// TwinCAT 3 PLC project Nepionic_Log_Test
// ProgramVersion: 3.1.4026.22
// libraries:
//   [Nepionic_Log], * (Nepionic)
//   [Nepionic_Log_OTel], * (Nepionic)
//   [Nepionic_Log_Syslog], * (Nepionic)
//   Tc2_Standard, * (Beckhoff Automation GmbH)
//   Tc2_System, * (Beckhoff Automation GmbH)
//   Tc2_Utilities, * (Beckhoff Automation GmbH)
//   TcUnit, * (www.tcunit.org)
//   Tc3_Module, * (Beckhoff Automation GmbH)
// project tree:
//   Lib/ LogTester.TcPOU (not stored)
//   Tests/ FB_Test_OTelLogAppender.TcPOU
//   Programs/ TestRunner.TcPOU
//   Tasks/ TestTask.TcTTO (not stored)
// real-time tasks:
//   TASK TestTask: cycle T#10ms, priority 20, ADS port 350

// ---- Tests/FB_Test_OTelLogAppender.TcPOU
/// TcUnit tests for OTelLogAppender.
/// Exercises ring slot writes, head advancement, sequence tagging,
/// severity mapping, attribute storage, ring wrap, and overflow counter.
FUNCTION_BLOCK FB_Test_OTelLogAppender EXTENDS TcUnit.FB_TestSuite
VAR
END_VAR

Test_HeadIncrements();
Test_SequenceCommitted();
Test_SlotContents();
Test_SeverityMapping();
Test_SlotAttrs();
Test_SlotIndexWraps();
Test_OverflowCnt();
Test_LevelProperty();

// head advances by 1 after a single Append call.
METHOD PRIVATE Test_HeadIncrements
VAR_INPUT END_VAR
VAR
	appender   : Nepionic_Log_OTel.OTelLogAppender;
	emptyAttrs : ARRAY[0..9] OF Nepionic_Log.LogAttribute;
END_VAR
TcUnit.Test('HeadIncrements');

appender.Append(Nepionic_Log.LogLevel.Information, 'hello', 'src', emptyAttrs, 0);

AssertEquals_UDINT(Expected := 1,
                   Actual   := appender.ring.head,
                   Message  := 'head should be 1 after one Append call');

TcUnit.Test_Finished();
END_METHOD

// Level property defaults to Debug; can be raised and read back.
METHOD PRIVATE Test_LevelProperty
VAR_INPUT END_VAR
VAR
	appender : Nepionic_Log_OTel.OTelLogAppender;
END_VAR
TcUnit.Test('LevelProperty');

AssertEquals_INT(Expected := Nepionic_Log.LogLevel.Debug,
                 Actual   := appender.Level,
                 Message  := 'default Level should be Debug');

appender.Level := Nepionic_Log.LogLevel.Warning;

AssertEquals_INT(Expected := Nepionic_Log.LogLevel.Warning,
                 Actual   := appender.Level,
                 Message  := 'Level should reflect the assigned value');

TcUnit.Test_Finished();
END_METHOD

// overflow_cnt must be 0 after the first full lap and 1 after the first wrap.
METHOD PRIVATE Test_OverflowCnt
VAR_INPUT END_VAR
VAR
	appender   : Nepionic_Log_OTel.OTelLogAppender;
	emptyAttrs : ARRAY[0..9] OF Nepionic_Log.LogAttribute;
	i          : UDINT;
END_VAR
TcUnit.Test('OverflowCnt');

// First 128 writes — slot_idx=0 at head=0 is guarded by head>0 check.
FOR i := 0 TO 127 DO
	appender.Append(Nepionic_Log.LogLevel.Debug, 'fill', 'src', emptyAttrs, 0);
END_FOR

AssertEquals_UDINT(Expected := 0,
                   Actual   := appender.ring.overflow_cnt,
                   Message  := 'overflow_cnt should be 0 after first 128 writes');

// 129th write: head=128, slot_idx=0, head>0 → overflow_cnt increments
appender.Append(Nepionic_Log.LogLevel.Debug, 'wrap', 'src', emptyAttrs, 0);

AssertEquals_UDINT(Expected := 1,
                   Actual   := appender.ring.overflow_cnt,
                   Message  := 'overflow_cnt should be 1 after first ring wrap');

TcUnit.Test_Finished();
END_METHOD

// After the first Append (absIdx=0, capacity=128):
//   expectedGen = (0/128 + 1)*2 = 2
// Slot 0 sequence must be 2 (EVEN = committed).
METHOD PRIVATE Test_SequenceCommitted
VAR_INPUT END_VAR
VAR
	appender   : Nepionic_Log_OTel.OTelLogAppender;
	emptyAttrs : ARRAY[0..9] OF Nepionic_Log.LogAttribute;
END_VAR
TcUnit.Test('SequenceCommitted');

appender.Append(Nepionic_Log.LogLevel.Information, 'hello', 'src', emptyAttrs, 0);

AssertEquals_UDINT(Expected := 2,
                   Actual   := appender.ring.entries[0].sequence,
                   Message  := 'sequence should be 2 (committed, generation 1)');

TcUnit.Test_Finished();
END_METHOD

// Each LogLevel maps to the correct numeric severity in the ring slot.
METHOD PRIVATE Test_SeverityMapping
VAR_INPUT END_VAR
VAR
	appender   : Nepionic_Log_OTel.OTelLogAppender;
	emptyAttrs : ARRAY[0..9] OF Nepionic_Log.LogAttribute;
END_VAR
TcUnit.Test('SeverityMapping');

// Write one entry per level; they land in consecutive slots 0..4.
appender.Append(Nepionic_Log.LogLevel.Debug,       'dbg',   '', emptyAttrs, 0);
appender.Append(Nepionic_Log.LogLevel.Information, 'info',  '', emptyAttrs, 0);
appender.Append(Nepionic_Log.LogLevel.Warning,     'warn',  '', emptyAttrs, 0);
appender.Append(Nepionic_Log.LogLevel.Error,       'err',   '', emptyAttrs, 0);
appender.Append(Nepionic_Log.LogLevel.Fatal,       'fatal', '', emptyAttrs, 0);

AssertEquals_UDINT(Expected := 0, Actual := appender.ring.entries[0].severity, Message := 'Debug should map to 0');
AssertEquals_UDINT(Expected := 1, Actual := appender.ring.entries[1].severity, Message := 'Information should map to 1');
AssertEquals_UDINT(Expected := 2, Actual := appender.ring.entries[2].severity, Message := 'Warning should map to 2');
AssertEquals_UDINT(Expected := 3, Actual := appender.ring.entries[3].severity, Message := 'Error should map to 3');
AssertEquals_UDINT(Expected := 4, Actual := appender.ring.entries[4].severity, Message := 'Fatal should map to 4');

TcUnit.Test_Finished();
END_METHOD

// attribute_count and key/value of populated attributes are stored correctly.
METHOD PRIVATE Test_SlotAttrs
VAR_INPUT END_VAR
VAR
	appender   : Nepionic_Log_OTel.OTelLogAppender;
	testAttrs  : ARRAY[0..9] OF Nepionic_Log.LogAttribute;
END_VAR
TcUnit.Test('SlotAttrs');

testAttrs[0].key       := 'batch.id';
testAttrs[0].attr_type := Nepionic_Log.LogAttributeType.Str;
// value_bytes: copy string 'BATCH-42' manually via assignment is not possible for byte arrays,
// but we can verify round-trip by checking key and attr_type at minimum.
testAttrs[1].key       := 'axis.speed';
testAttrs[1].attr_type := Nepionic_Log.LogAttributeType.Float64;

appender.Append(Nepionic_Log.LogLevel.Information, 'test', 'src', testAttrs, 2);

AssertEquals_UDINT(Expected := 2,
                   Actual   := appender.ring.entries[0].attribute_count,
                   Message  := 'attribute_count should be 2');

AssertEquals_STRING(Expected := 'batch.id',
                    Actual   := appender.ring.entries[0].attributes[0].key,
                    Message  := 'attrs[0].key mismatch');

AssertEquals_STRING(Expected := 'axis.speed',
                    Actual   := appender.ring.entries[0].attributes[1].key,
                    Message  := 'attrs[1].key mismatch');

TcUnit.Test_Finished();
END_METHOD

// message, source, and attribute_count are stored correctly.
METHOD PRIVATE Test_SlotContents
VAR_INPUT END_VAR
VAR
	appender   : Nepionic_Log_OTel.OTelLogAppender;
	emptyAttrs : ARRAY[0..9] OF Nepionic_Log.LogAttribute;
END_VAR
TcUnit.Test('SlotContents');

appender.Append(Nepionic_Log.LogLevel.Warning, 'Drive fault detected', 'MAIN.AxisX', emptyAttrs, 0);

AssertEquals_STRING(Expected := 'Drive fault detected',
                    Actual   := appender.ring.entries[0].message,
                    Message  := 'message mismatch');

AssertEquals_STRING(Expected := 'MAIN.AxisX',
                    Actual   := appender.ring.entries[0].source,
                    Message  := 'source mismatch');

AssertEquals_UDINT(Expected := 0,
                   Actual   := appender.ring.entries[0].attribute_count,
                   Message  := 'attribute_count should be 0');

TcUnit.Test_Finished();
END_METHOD

// After 128 writes the ring wraps: the 129th Append targets slot 0.
// entries[0].sequence must be 4 (generation 2) and message must be the new value.
METHOD PRIVATE Test_SlotIndexWraps
VAR_INPUT END_VAR
VAR
	appender   : Nepionic_Log_OTel.OTelLogAppender;
	emptyAttrs : ARRAY[0..9] OF Nepionic_Log.LogAttribute;
	i          : UDINT;
END_VAR
TcUnit.Test('SlotIndexWraps');

// Fill ring once (writes to slots 0..127, head advances to 128)
FOR i := 0 TO 127 DO
	appender.Append(Nepionic_Log.LogLevel.Debug, 'fill', 'src', emptyAttrs, 0);
END_FOR

AssertEquals_UDINT(Expected := 128,
                   Actual   := appender.ring.head,
                   Message  := 'head should be 128 after 128 writes');

// 129th write: slot_idx = 128 MOD 128 = 0 → overwrites slot 0
appender.Append(Nepionic_Log.LogLevel.Information, 'wrapped', 'src', emptyAttrs, 0);

AssertEquals_UDINT(Expected := 129,
                   Actual   := appender.ring.head,
                   Message  := 'head should be 129 after 129th write');

AssertEquals_STRING(Expected := 'wrapped',
                    Actual   := appender.ring.entries[0].message,
                    Message  := 'slot 0 should be overwritten by the 129th write');

// expectedGen = (128 / 128 + 1) * 2 = 4
AssertEquals_UDINT(Expected := 4,
                   Actual   := appender.ring.entries[0].sequence,
                   Message  := 'sequence at slot 0 should be 4 (generation 2)');

TcUnit.Test_Finished();
END_METHOD

END_FUNCTION_BLOCK

// ---- Programs/TestRunner.TcPOU
PROGRAM TestRunner
VAR
	ads_log_appender : AdsLogAppender;
	syslog_appender : SyslogAppender(hostname := '127.0.0.1', port := 514);
	otel_log_appender : OTelLogAppender;
	logger : DefaultLogger('TestRunner');
	fbTestOTelLogAppender : FB_Test_OTelLogAppender;
	
	get_local_ams_netid : Tc2_Utilities.Fb_GetLocalAmsNetId;
	
	initialised : BOOL;
	
	message : STRING(255) := 'We modded with 100 nicely!';
	
	some_incrementing_value : UDINT;
	
	yeah_boi : BOOL;
	log_tester : LogTester;
END_VAR

IF NOT initialised THEN
	get_local_ams_netid(bExecute := TRUE);
	
	IF NOT get_local_ams_netid.bBusy THEN
		get_local_ams_netid(bExecute := FALSE);
		GetLogManager().Register(ads_log_appender);
		GetLogManager().Register(syslog_appender);
		GetLogManager().Register(otel_log_appender);
		initialised := TRUE;
	END_IF
END_IF

IF some_incrementing_value MOD 100 = 0 THEN
	logger
		.WithAttribute('ams-netid', get_local_ams_netid.AddrString)
		.WithUDintAttribute('some_incrementing_value', some_incrementing_value)
		.Info(message);
END_IF

some_incrementing_value := some_incrementing_value + 1;

IF yeah_boi THEN
	yeah_boi := FALSE;
	log_tester.YeahBoi();
END_IF

syslog_appender.Execute();
fbTestOTelLogAppender();

END_PROGRAM
